(* CoDeSys 2.3 export: ST_PSX_VALVE_IN.EXP *)

(* Data type *)
TYPE ST_PSX_VALVE_IN :
STRUCT
	Status : UINT;
	Actual : INT;
	Error  : UINT;

END_STRUCT
END_TYPE
